/// doc
PROGRAM MAIN
VAR
  _variant : STRING := 'Default';
  _firstCycle : BOOL := TRUE;
  _pushover : Pushover.PushoverClient('my-token', 'my-user');
  _message : STRING(255);
  _unusedButLoved : INT;
END_VAR

IF _firstCycle
THEN
  _firstCycle := FALSE;
  _message := CONCAT(CONCAT('Application using variant ', _variant), ' started');
  _pushover.SendMessageAsync('MyApplication', _message);
END_IF

_pushover.Cyclic();

END_PROGRAM

(* stored: Version 1.1.0.1, ProductVersion 3.1.4026.12
   POU MAIN: Id {aa34fcfe-6c3e-4d22-9edb-c207d34b0a3c}, SpecialFunc None *)
